(* CODESYS project FirstSteps.project

Project tree, tasks and I/O mapping:
  Device : CODESYS Control for Raspberry Pi SL, 3S - Smart Software Solutions GmbH, version 3.5.12.30
    application Application
      libraries: AC_ModuleBase, 3.5.0.0 (3S - Smart Software Solutions GmbH); Standard, 3.5.12.0 (System)
      task AC_RMP_Task (cyclic, interval t#20ms, priority 30) calls AC_PRG_RMP
      task STANDARD (cyclic, interval t#10ms, priority 5) calls AC_CALL_STANDARD_START, AC_CALL_STANDARD_END
      global variables GVL_Simulation_I_O
      AC_Std/
        global variables GVL_Room
        global variables MODULE_INFOS
        global variables GVL_MODULE_TREE
        function AC_InitInternal [ST]
        function AC_Init [ST]
        function AC_OnlineChange [ST]
        function AC_Io_ChannelRefCode_STANDARD [ST]
        program AC_CALL_STANDARD_START [ST]
        program AC_CALL_STANDARD_END [ST]
      AC_FBs/
        function block AC_Room_Light1 [ST]
        function block AC_Room_LightSimple1 [ST]
        function block AC_Room_Light2 [ST]
        function block AC_Room [ST]
      AC_RMP/
        global variables AC_RMP
        program AC_PRG_RMP [ST]
    SoftMotion General Axis Pool
    I²C
    SPI
      SPI_master : SPI master, 3S - Smart Software Solutions GmbH, version 1.0.0.0
          settings: _diBitsPerWord = 8; _diMaxSpeed = 1000000
        Monarco_HAT : Monarco HAT, Monarco.io, version 2.0.0.0
            input  Application.GVL_Room.Room.INST_Light1.INST_Switch.xIn : BOOL  // DigIn.Bit0
            input  Application.GVL_Room.Room.INST_LightSimple1.INST_SwitchSimple.xIn : BOOL  // DigIn.Bit1
            input  Application.GVL_Room.Room.INST_Light2.INST_Switch.xIn : BOOL  // DigIn.Bit2
            output Application.GVL_Room.Room.INST_LightSimple1.xSwitchedOn : BOOL  // DigOut.Bit0
            output Application.GVL_Room.Room.INST_Light1.uiBrightness : WORD  // AO0
            output Application.GVL_Room.Room.INST_Light2.uiBrightness : WORD  // AO1
            unmapped channels: DigIn, AI0, AI1, DigOut
    GPIOs_A_B : GPIOs A/B, 3S - Smart Software Solutions GmbH, version 3.5.11.0
        unmapped channels: digital inputs (GPIO0..GPIO31), digital outputs (GPIO0..GPIO31)
    Onewire
    Camera device
      <Empty>
  libraries: AC_ModuleBase, 3.5.0.0 (3S - Smart Software Solutions GmbH)
  5ce3da45-db07-42e7-a21c-a00fff4ed8f6|D:\Libraries\trunk\Application\ApplicationComposer\AC_Building\0.34.3.5 draft\floor32.bmp
  5ce3da45-db07-42e7-a21c-a00fff4ed8f6|C:\Users\Public\Pictures\Sample Pictures\Chrysanthemum.jpg
  5ce3da45-db07-42e7-a21c-a00fff4ed8f6|C:\Users\Public\Pictures\Sample Pictures\Desert.jpg
  Room
    Lights (Lights)
      Light2
        Switch (Switch)
        Switch
      LightSimple1
        SwitchSimple
        Switch (SwitchSimple)
      Light1
        Switch (Switch)
        Switch
  AC_GENERATOR_DATA
  5ce3da45-db07-42e7-a21c-a00fff4ed8f6|C:\Users\b.joedicke\Pictures\light_16.png
  5ce3da45-db07-42e7-a21c-a00fff4ed8f6|C:\Users\b.joedicke\Pictures\light_32.png
  5ce3da45-db07-42e7-a21c-a00fff4ed8f6|C:\Users\b.joedicke\Pictures\room16.bmp
  5ce3da45-db07-42e7-a21c-a00fff4ed8f6|C:\Users\b.joedicke\Pictures\room32.bmp
  5ce3da45-db07-42e7-a21c-a00fff4ed8f6|C:\Users\b.joedicke\Pictures\switch_16.png
  5ce3da45-db07-42e7-a21c-a00fff4ed8f6|C:\Users\b.joedicke\Pictures\switch_32.png
  5ce3da45-db07-42e7-a21c-a00fff4ed8f6|C:\Users\b.joedicke\Pictures\switchsimple_32.png
  5ce3da45-db07-42e7-a21c-a00fff4ed8f6|C:\room16.bmp
  5ce3da45-db07-42e7-a21c-a00fff4ed8f6|C:\Users\b.joedicke\Pictures\lightsimple_16.png
  5ce3da45-db07-42e7-a21c-a00fff4ed8f6|C:\switchsimple_16.png
  5ce3da45-db07-42e7-a21c-a00fff4ed8f6|C:\Users\b.joedicke\Pictures\switchsimple_16.png
  5ce3da45-db07-42e7-a21c-a00fff4ed8f6|C:\Users\b.joedicke\Pictures\lightsimple_32.png
  5ce3da45-db07-42e7-a21c-a00fff4ed8f6|D:\Libraries\trunk\Application\ApplicationComposer\AC_Building\0.34.3.5 draft\SwitchOnOff32.ico
  5ce3da45-db07-42e7-a21c-a00fff4ed8f6|C:\light_16.png
  5ce3da45-db07-42e7-a21c-a00fff4ed8f6|C:\light_32.png
  5ce3da45-db07-42e7-a21c-a00fff4ed8f6|D:\Libraries\trunk\Application\ApplicationComposer\AC_Building\0.34.3.5 draft\LightStandard16.ico
  5ce3da45-db07-42e7-a21c-a00fff4ed8f6|D:\Libraries\trunk\Application\ApplicationComposer\AC_Building\0.34.3.5 draft\LightStandard32.bmp
  5ce3da45-db07-42e7-a21c-a00fff4ed8f6|D:\Libraries\trunk\Application\ApplicationComposer\AC_Building\0.34.3.5 draft\LightStandard32.ico
  5ce3da45-db07-42e7-a21c-a00fff4ed8f6|D:\Libraries\trunk\Application\ApplicationComposer\AC_Building\0.34.3.5 draft\LightDimmed16.ico
  5ce3da45-db07-42e7-a21c-a00fff4ed8f6|D:\Libraries\trunk\Application\ApplicationComposer\AC_Building\0.34.3.5 draft\LightDimmed32.ico
  5ce3da45-db07-42e7-a21c-a00fff4ed8f6|D:\Libraries\trunk\Application\ApplicationComposer\AC_Building\0.34.3.5 draft\room16.bmp
  5ce3da45-db07-42e7-a21c-a00fff4ed8f6|D:\Libraries\trunk\Application\ApplicationComposer\AC_Building\0.34.3.5 draft\room32.bmp
  5ce3da45-db07-42e7-a21c-a00fff4ed8f6|D:\Libraries\trunk\Application\ApplicationComposer\AC_Building\0.34.3.5 draft\SwitchPush16.ico
  5ce3da45-db07-42e7-a21c-a00fff4ed8f6|D:\Libraries\trunk\Application\ApplicationComposer\AC_Building\0.34.3.5 draft\SwitchPush32.ico
  5ce3da45-db07-42e7-a21c-a00fff4ed8f6|D:\Libraries\trunk\Application\ApplicationComposer\AC_Building\0.34.3.5 draft\SwitchOnOff16.ico
  Room/
    text Room
    function block Room [ST]
    text list TL
    Light/
      interface ILight
      text Light
      function block Light [ST]: CallPrioMediumStart
      text LightSimple
      function block LightSimple [ST]: CallPrioMediumStart
    Switch/
      text Switch
      interface ISwitch: Push, PushLong
      function block Switch [ST]: Push, PushLong, CallPrioMediumStart
      interface ISwitchSimple: On
      text SwitchSimple
      function block SwitchSimple [ST]: On
    image pool IP
  5ce3da45-db07-42e7-a21c-a00fff4ed8f6|D:\Libraries\trunk\Application\ApplicationComposer\AC_Building\0.34.3.5 draft\room16.bmp
  5ce3da45-db07-42e7-a21c-a00fff4ed8f6|D:\Libraries\trunk\Application\ApplicationComposer\AC_Building\0.34.3.5 draft\room32.bmp
  5ce3da45-db07-42e7-a21c-a00fff4ed8f6|D:\Libraries\trunk\Application\ApplicationComposer\AC_Building\0.34.3.5 draft\SwitchPush16.ico
  5ce3da45-db07-42e7-a21c-a00fff4ed8f6|D:\Libraries\trunk\Application\ApplicationComposer\AC_Building\0.34.3.5 draft\SwitchPush32.ico
  5ce3da45-db07-42e7-a21c-a00fff4ed8f6|D:\Libraries\trunk\Application\ApplicationComposer\AC_Building\0.34.3.5 draft\LightDimmed16.ico
  5ce3da45-db07-42e7-a21c-a00fff4ed8f6|D:\Libraries\trunk\Application\ApplicationComposer\AC_Building\0.34.3.5 draft\LightDimmed32.ico
  5ce3da45-db07-42e7-a21c-a00fff4ed8f6|D:\Libraries\trunk\Application\ApplicationComposer\AC_Building\0.34.3.5 draft\LightStandard16.ico
  5ce3da45-db07-42e7-a21c-a00fff4ed8f6|D:\Libraries\trunk\Application\ApplicationComposer\AC_Building\0.34.3.5 draft\LightStandard32.ico
  5ce3da45-db07-42e7-a21c-a00fff4ed8f6|D:\Libraries\trunk\Application\ApplicationComposer\AC_Building\0.34.3.5 draft\SwitchOnOff16.ico
  5ce3da45-db07-42e7-a21c-a00fff4ed8f6|D:\Libraries\trunk\Application\ApplicationComposer\AC_Building\0.34.3.5 draft\SwitchOnOff32.ico
*)

// Device/Application/GVL_Simulation_I_O
VAR_GLOBAL

//these variables are normally real inputs and outputs. 
///For simulation reason, they are declared here and can be used to test the app.	

	xPushSwitch			: BOOL;
	xPushSimpleSwitch	: BOOL;

	uiBrightness		: UINT;
	xSimpleOn			: BOOL;
END_VAR

// Device/Application/AC_Std/GVL_Room
//Code generated by Application Composer.
//Modifying generated code is not recommended!

VAR_GLOBAL
	Room: AC_Room;
END_VAR

// Device/Application/AC_Std/MODULE_INFOS
//Code generated by Application Composer.
//Modifying generated code is not recommended!
{attribute 'global_init_slot' := '40000'}
{attribute 'init_on_onlchange'}

VAR_GLOBAL
	{attribute 'init_on_onlchange'}
	Room_INFO: AC.ModuleInfo := (pbyModuleType := ADR('Room'));
	{attribute 'init_on_onlchange'}
	Light_INFO: AC.ModuleInfo := (pbyModuleType := ADR('Light'));
	{attribute 'init_on_onlchange'}
	LightSimple_INFO: AC.ModuleInfo := (pbyModuleType := ADR('LightSimple'));
	{attribute 'init_on_onlchange'}
	Switch_INFO: AC.ModuleInfo := (pbyModuleType := ADR('Switch'));
	{attribute 'init_on_onlchange'}
	SwitchSimple_INFO: AC.ModuleInfo := (pbyModuleType := ADR('SwitchSimple'));
END_VAR

// Device/Application/AC_Std/GVL_MODULE_TREE
//Code generated by Application Composer.
//Modifying generated code is not recommended!

VAR_GLOBAL
	Module_Tree: AC.ModuleTree;
	aNodes: ARRAY[0..7] OF AC.MNode;
	AC_Environment: AC.MEnv;
END_VAR

// Device/Application/AC_RMP/AC_RMP
//Code generated by Application Composer.
//Modifying generated code is not recommended!
{attribute 'global_init_slot' := '60000'}
{attribute 'init_on_onlchange'}

VAR_GLOBAL
	{attribute 'init_on_onlchange'}
	AC_RMP_Service: AC.RMPService := (uiLocalAppID:=9744, uiNumberOfConnections:=0, pSendConnection:=0, pReceiveConnection:=0);
END_VAR

// Device/Application/AC_RMP/AC_PRG_RMP
//Code generated by Application Composer.
//Modifying generated code is not recommended!
PROGRAM AC_PRG_RMP
VAR
    itfRmpService2 : AC.IRmpService2 := 0;
    xStartCyclicAction : BOOL;
    xIsActionOngoing : BOOL;
    xValid : BOOL;
    xValidEnd : BOOL := TRUE;
END_VAR

//Code generated by Application Composer.
//Modifying generated code is not recommended!
__QUERYINTERFACE(AC_RMP_Service, itfRmpService2);
IF itfRmpService2 <> 0 AND xValidEnd THEN
    xValid := itfRmpService2.GetIsActionOngoing(xIsActionOngoing=>xIsActionOngoing);
    IF NOT xValid OR (xValid AND xIsActionOngoing) THEN
        xStartCyclicAction := FALSE;
    ELSE
        xStartCyclicAction := itfRmpService2.SetIsActionOngoing(TRUE);
    END_IF
ELSE
    xStartCyclicAction := TRUE;
END_IF
IF xStartCyclicAction THEN
    AC_RMP_Service.CyclicCall() ;
END_IF
IF itfRmpService2 <> 0 AND (xStartCyclicAction OR NOT xValidEnd) THEN
    xValidEnd := itfRmpService2.SetIsActionOngoing(FALSE);
END_IF

END_PROGRAM

// Device/Application/AC_Std/AC_CALL_STANDARD_START
//Code generated by Application Composer.
//Modifying generated code is not recommended!
PROGRAM AC_CALL_STANDARD_START

//Code generated by Application Composer.
//Modifying generated code is not recommended!
AC_Io_ChannelRefCode_STANDARD() ;
Room.CallPrioMEDIUMStart() ;

END_PROGRAM

// Device/Application/AC_Std/AC_Io_ChannelRefCode_STANDARD
//Code generated by Application Composer.
//Modifying generated code is not recommended!
FUNCTION AC_Io_ChannelRefCode_STANDARD

//Code generated by Application Composer.
//Modifying generated code is not recommended!

//Special code to make sure mapped I/O variables are updated in the correct task

{IF defined(variable:Application.GVL_Room.Room.INST_Light1.uiBrightness) AND defined(variable:Application.GVL_Room.Room.INST_LightSimple1.xSwitchedOn) AND defined(variable:Application.GVL_Room.Room.INST_Light2.uiBrightness) AND defined(variable:Application.GVL_Room.Room.INST_Light1.INST_Switch.xIn) AND defined(variable:Application.GVL_Room.Room.INST_LightSimple1.INST_SwitchSimple.xIn) AND defined(variable:Application.GVL_Room.Room.INST_Light2.INST_Switch.xIn)}
 ;
{END_IF}

END_FUNCTION

// Room/Room
FUNCTION_BLOCK Room EXTENDS AC.Module
VAR_INPUT
	//Submodule Lights
	pLights				: POINTER TO ILight;
	uiNumberOfLights	: UINT;
END_VAR
VAR_OUTPUT
END_VAR
VAR
END_VAR

END_FUNCTION_BLOCK

// Room/Light/ILight
INTERFACE ILight EXTENDS AC.IModule

END_INTERFACE

// Device/Application/AC_Std/AC_CALL_STANDARD_END
//Code generated by Application Composer.
//Modifying generated code is not recommended!
PROGRAM AC_CALL_STANDARD_END

//Code generated by Application Composer.
//Modifying generated code is not recommended!
Room.CallPrioMEDIUMEnd() ;

END_PROGRAM

// Room/Light/Light
FUNCTION_BLOCK Light EXTENDS AC.Module IMPLEMENTS ILight
VAR_INPUT
	//Submodule Switch
	Switch		: ISwitch;
	
	//parameter
	uiMaxValue	: UINT := 5000 ;
	rSpeed	: REAL := 25; //percentage per second
END_VAR
VAR_OUTPUT
	uiBrightness	: UINT;
END_VAR
VAR
	rPercentageOn	: REAL; (* percentage from 0 to 1 *)
	tTaskCycle		: TIME := T#10MS;
	rDirection		: REAL := 1; (* 1 --> switch the light on --> switch it off *)
	
	xChangeDirection: BOOL; (* helper variable *)
	xChangeDirectionPush: BOOL; (* helper variable *)
	
	iState			: INT;
END_VAR

(* Called at the start of the medium priority task if one is defined.
 Note: the return value is not used.*)
METHOD CallPrioMediumStart : BOOL
VAR
	pModule: POINTER TO AC.Module;
END_VAR
SUPER^.CallPrioMediumStart();

CASE iState OF
	
	0: (* check the state of the switch *)
		IF Switch.PushLong THEN
			xChangeDirection := TRUE;
			iState := 10;
		ELSIF NOT Switch.PushLong AND xChangeDirection THEN
			xChangeDirection := FALSE;
			iState := 20;
			
		ELSIF Switch.Push THEN
			iState := 30;
			xChangeDirectionPush := TRUE;
			
		ELSIF NOT Switch.Push AND xChangeDirectionPush THEN
			xChangeDirectionPush := FALSE;
			iState := 20;
		END_IF
	
	10: (* dim function *)
		rPercentageOn := rPercentageOn + rDirection * rSpeed * TIME_TO_REAL(tTaskCycle)/100000;
		IF rPercentageOn > 1 THEN
			rPercentageOn := 1;
			
		ELSIF rPercentageOn < 0 THEN
			rPercentageOn := 0;
		END_IF
		iState := 0;
	
	20: (* check if the direction must be changed *)
		IF rDirection = 1 AND rPercentageOn = 1 THEN
			rDirection := -1;
		ELSIF
			rDirection = -1 AND rPercentageOn = 0 THEN
			rDirection := 1;
		END_IF
		iState := 0;
	
	30:(* invert light *)
		IF rPercentageOn = 1 THEN
			rPercentageOn :=0;
		ELSE
			rPercentageOn := 1;
		END_IF
		iState := 0;

END_CASE

uiBrightness := REAL_TO_UINT(rPercentageOn*uiMaxValue);
END_METHOD

END_FUNCTION_BLOCK

// Room/Switch/Switch
FUNCTION_BLOCK Switch EXTENDS AC.Module IMPLEMENTS ISwitch
VAR_INPUT
	// Input
	xIn		: BOOL;
	//parameter
	tTimer	: TIME := T#500MS;
END_VAR

VAR
	timerLong	: TON; (* timer to know how long the switch is tapped *)
	
	xPush	: BOOL; (* signal to toggle the light *)
	xPushLong : BOOL; (* signal to dim the light *)
	
	iState	: INT;
END_VAR

PROPERTY PUBLIC Push : BOOL
GET
Push := xPush;
END_GET
END_PROPERTY

PROPERTY PUBLIC PushLong : BOOL
GET
PushLong := xPushLong;
END_GET
END_PROPERTY

(* Called at the start of the medium priority task if one is defined.
 Note: the return value is not used.*)
METHOD CallPrioMediumStart : BOOL
SUPER^.CallPrioMediumStart();

xPush := FALSE;

CASE iState OF
	0: (* initialization *)
		xPush := xPushLong := FALSE;
		IF NOT xIn THEN
			iState := 10;
		END_IF
		
	10: (* switch is pushed *)
		IF xIn THEN
			iState := 20;
			timerLong(IN := FALSE, PT := tTimer);
		END_IF

	20: (* timer is started, to check if the toggle or dim function should be used *)
		timerLong(IN := TRUE);
		IF NOT xIn THEN
			xPush := TRUE;
			iState := 0;
		ELSIF timerLong.Q THEN
			iState := 30;
		END_IF
		
	30: (* the dim function is used *)
		xPushLong := TRUE;
		IF NOT xIn THEN
			iState := 0;
		END_IF
		

END_CASE
END_METHOD

END_FUNCTION_BLOCK

// Room/Switch/ISwitch
INTERFACE ISwitch IMPLEMENTS AC.IModule

PROPERTY Push : BOOL
GET
END_GET
END_PROPERTY

PROPERTY PushLong : BOOL
GET
END_GET
END_PROPERTY

END_INTERFACE

// Room/Light/LightSimple
FUNCTION_BLOCK LightSimple EXTENDS AC.Module IMPLEMENTS ILight
VAR_INPUT
	// Submodule Switch
	SwitchSimple	: ISwitchSimple;
END_VAR
VAR_OUTPUT
	xSwitchedOn		: BOOL;
END_VAR
VAR
END_VAR

(* Called at the start of the medium priority task if one is defined.
 Note: the return value is not used.*)
METHOD CallPrioMediumStart : BOOL
SUPER^.CallPrioMediumStart();

xSwitchedOn := SwitchSimple.On;
END_METHOD

END_FUNCTION_BLOCK

// Room/Switch/SwitchSimple
FUNCTION_BLOCK SwitchSimple EXTENDS AC.Module IMPLEMENTS ISwitchSimple
VAR_INPUT
	// Input
	xIn		: BOOL;
END_VAR
VAR_OUTPUT
END_VAR
VAR
	xOn	: BOOL;
END_VAR

PROPERTY PUBLIC On : BOOL
GET
On := xIn;
END_GET
END_PROPERTY

END_FUNCTION_BLOCK

// Room/Switch/ISwitchSimple
INTERFACE ISwitchSimple IMPLEMENTS AC.IModule

PROPERTY On : BOOL
GET
END_GET
END_PROPERTY

END_INTERFACE

// Device/Application/AC_FBs/AC_Room_Light1
//Code generated by Application Composer.
//Modifying generated code is not recommended!
FUNCTION_BLOCK AC_Room_Light1 EXTENDS Light
VAR_INPUT 
    INST_Switch : Switch;
END_VAR

//Code generated by Application Composer.
//Modifying generated code is not recommended!
SUPER^();

END_FUNCTION_BLOCK

// Device/Application/AC_FBs/AC_Room_LightSimple1
//Code generated by Application Composer.
//Modifying generated code is not recommended!
FUNCTION_BLOCK AC_Room_LightSimple1 EXTENDS LightSimple
VAR_INPUT 
    INST_SwitchSimple : SwitchSimple;
END_VAR

//Code generated by Application Composer.
//Modifying generated code is not recommended!
SUPER^();

END_FUNCTION_BLOCK

// Device/Application/AC_FBs/AC_Room_Light2
//Code generated by Application Composer.
//Modifying generated code is not recommended!
FUNCTION_BLOCK AC_Room_Light2 EXTENDS Light
VAR_INPUT 
    INST_Switch : Switch;
END_VAR

//Code generated by Application Composer.
//Modifying generated code is not recommended!
SUPER^();

END_FUNCTION_BLOCK

// Device/Application/AC_FBs/AC_Room
//Code generated by Application Composer.
//Modifying generated code is not recommended!
FUNCTION_BLOCK AC_Room EXTENDS Room
VAR_INPUT 
    INST_Light1 : AC_Room_Light1;
    INST_LightSimple1 : AC_Room_LightSimple1;
    INST_Light2 : AC_Room_Light2;
    AC_ARRAY_pLights : ARRAY[0..2] OF ILight;
END_VAR

//Code generated by Application Composer.
//Modifying generated code is not recommended!
SUPER^();

END_FUNCTION_BLOCK

// Device/Application/AC_Std/AC_InitInternal
//Code generated by Application Composer.
//Modifying generated code is not recommended!
FUNCTION AC_InitInternal
VAR_INPUT
  bOnlineChange : BOOL ;
END_VAR
VAR
  hnd : AC.ModuleHandle ;
END_VAR

//Code generated by Application Composer.
//Modifying generated code is not recommended!
AC_Environment.mtree := Module_Tree ;
AC_Environment.rmps := AC_RMP_Service ;
{IF defined(variable:AC_Environment.exts)}
	AC_Environment.exts := 0 ;
	AC_Environment.uiexts := 0 ;
{END_IF}
Module_Tree.Init(ADR(aNodes), 8);
hnd := Module_Tree.AddChild(0, Room);
Room.SetIdentification(ADR('Room'), ADR(Room_INFO), 16#2610A9CF, hnd, ADR(AC_Environment)) ;
hnd := Module_Tree.AddChild(Room, Room.INST_Light2);
Room.INST_Light2.SetIdentification(ADR('Light2'), ADR(Light_INFO), 16#26100F2D, hnd, ADR(AC_Environment)) ;
hnd := Module_Tree.AddChild(Room, Room.INST_LightSimple1);
Room.INST_LightSimple1.SetIdentification(ADR('LightSimple1'), ADR(LightSimple_INFO), 16#2610E8D4, hnd, ADR(AC_Environment)) ;
hnd := Module_Tree.AddChild(Room, Room.INST_Light1);
Room.INST_Light1.SetIdentification(ADR('Light1'), ADR(Light_INFO), 16#2610C045, hnd, ADR(AC_Environment)) ;
hnd := Module_Tree.AddChild(Room.INST_Light2, Room.INST_Light2.INST_Switch);
Room.INST_Light2.INST_Switch.SetIdentification(ADR('Switch'), ADR(Switch_INFO), 16#261067C5, hnd, ADR(AC_Environment)) ;
hnd := Module_Tree.AddChild(Room.INST_LightSimple1, Room.INST_LightSimple1.INST_SwitchSimple);
Room.INST_LightSimple1.INST_SwitchSimple.SetIdentification(ADR('SwitchSimple'), ADR(SwitchSimple_INFO), 16#26107A30, hnd, ADR(AC_Environment)) ;
hnd := Module_Tree.AddChild(Room.INST_Light1, Room.INST_Light1.INST_Switch);
Room.INST_Light1.INST_Switch.SetIdentification(ADR('Switch'), ADR(Switch_INFO), 16#2610E8FB, hnd, ADR(AC_Environment)) ;
Room.uiNumberOfLights := 3;
Room.AC_ARRAY_pLights[0] := Room.INST_Light1;
Room.AC_ARRAY_pLights[1] := Room.INST_LightSimple1;
Room.AC_ARRAY_pLights[2] := Room.INST_Light2;
Room.pLights := ADR(Room.AC_ARRAY_pLights);
Room.INST_Light1.Switch := Room.INST_Light1.INST_Switch;
Room.INST_LightSimple1.SwitchSimple := Room.INST_LightSimple1.INST_SwitchSimple;
Room.INST_Light2.Switch := Room.INST_Light2.INST_Switch;
IF bOnlineChange THEN
    Room.INST_Light1.uiMaxValue := 5000;
    Room.INST_Light1.rSpeed := 25;
    Room.INST_Light2.uiMaxValue := 5000;
    Room.INST_Light2.rSpeed := 25;
    Room.INST_Light1.INST_Switch.tTimer := TIME#500ms;
    Room.INST_Light2.INST_Switch.tTimer := TIME#500ms;
END_IF
Room.Init(bOnlineChange);

END_FUNCTION

// Device/Application/AC_Std/AC_Init
//Code generated by Application Composer.
//Modifying generated code is not recommended!
{attribute 'linkalways'}
{attribute 'call_after_global_init_slot' := '1234'}
FUNCTION AC_Init

//Code generated by Application Composer.
//Modifying generated code is not recommended!
AC_InitInternal(FALSE);

END_FUNCTION

// Device/Application/AC_Std/AC_OnlineChange
//Code generated by Application Composer.
//Modifying generated code is not recommended!
{attribute 'linkalways'}
{attribute 'call_after_online_change_slot' := '1234'}
FUNCTION AC_OnlineChange

//Code generated by Application Composer.
//Modifying generated code is not recommended!
Room.OnBeforeOnlineChange();
AC_InitInternal(TRUE);
Room.OnAfterOnlineChange();

END_FUNCTION

(* text list TL (id | default)
  Room_Desc | This is a room.
  UnitStandard_Task | This is a standard task.
  Role_Lights | Lights
  Light_Desc | This is a light, which can be dimmed and switched on and off.
  Switch_Desc | This is a switch, which has a tap and dim function.
  Light_Name_xOn | xOn
  Light_Desc_xOn | Licht eingeschalten (True) / ausgeschalten (False)
  Role_Switch | Switch
  Name_uiBrightness | Brightness
  Desc_uiBrightness | The brightness of the light.
  Name_uiMaxValue | maxLightValue
  Desc_uiMaxValue | The maximum value of the light.
  NAME_rSpeed | Speed
  DESC_rSpeed | The speed of the dimmer.
  NAME_tTimer | Timer
  DESC_tTimer | The time the switch has to wait before switching to the dim modus.
  Switch_Name_xIn | xIn
  Switch_Desc_xIn | Input of the Switch.
  SwitchSimple_Name_xIn | xIn (Simple)
  SwitchSimple_Desc_xIn | State of the switch (on / off)
  LightSimple_Desc | The simple light can be switched on and off.
  Name_switchedOn | SwitchedOn
  Desc_switchedOn | True, when the light is switched on and false when it is off.
  SwitchSimple_Desc | The simple switch has an on and off position.
   |  *)

(* text Room
MODULE Room IMPLEMENTED_BY Room
SEC MetaData
	Desc       := TL.Room_Desc ;
	Category   := 'FirstSteps' ;
	Icon_16    := IP.Room_Icon_16 ;
	Icon_32    := IP.Room_Icon_32 ;
END_SEC
SEC Toplevel
	GVL_name := 'GVL_%InstanceName%' ;
    SEC Standard_Task : MEDIUM
		Name  := STANDARD ;
		Desc  := TL.UnitStandard_Task ;
		Flags := CREATE_IF_MISSING | UPDATE_IOS ; ( * at least one task must use the "UPDATE_IOS" flag. * )
	END_SEC
END_SEC

SEC Slots
	SEC Slot_Multi	: Lights
		Variable	:= pLights;
		Var_Count	:= uiNumberOfLights;
		Role		:= TL.Role_Lights;
		Cardinality := [1..3];
		Type		:= SUBMODULE;
	END_SEC	
END_SEC
*)

(* text Light
MODULE Light IMPLEMENTED_BY Light
SEC MetaData
	Desc := TL.Light_Desc ;
	Category := 'FirstSteps' ;
	Icon_16 := IP.Light_Icon_16 ;
	Icon_32 := IP.Light_Icon_32 ;
END_SEC

SEC Slots
	SEC Slot : Switch
		Variable := Switch;
		Role := TL.Role_Switch;
		Type := SUBMODULE;
	END_SEC
END_SEC

SEC IO
	SEC Output : uiBrightness
		Variable := uiBrightness;
		Name := TL.Name_uiBrightness;
		Desc := TL.Desc_uiBrightness;
	END_SEC
END_SEC

SEC Parameters
	SEC Param : uiMaxValue
		Variable := uiMaxValue;
		Name := TL.Name_uiMaxValue;
		Desc := TL.Desc_uiMaxValue;
	END_SEC

	SEC Param : rSpeed
		Variable := rSpeed ;
		Name := TL.NAME_rSpeed ;
		Desc := TL.DESC_rSpeed ;
	END_SEC
END_SEC
*)

(* text LightSimple
MODULE LightSimple IMPLEMENTED_BY LightSimple
SEC MetaData
	Desc       := TL.LightSimple_Desc ;
	Category   := 'FirstSteps' ;
	Icon_16    := IP.LightSimple_Icon_16 ;
	Icon_32    := IP.LightSimple_Icon_32 ;
END_SEC

SEC Slots
	SEC Slot : SwitchSimple
		Variable := SwitchSimple;
		Role := TL.Role_Switch;
		Type := SUBMODULE;
	END_SEC
END_SEC

SEC IO
	SEC Output : SwitchedOn
		Variable := xSwitchedOn;
		Name := TL.Name_switchedOn;
		Desc := TL.Desc_switchedOn;
	END_SEC
END_SEC
*)

(* text Switch
MODULE Switch IMPLEMENTED_BY Switch
SEC MetaData
	Desc       := TL.Switch_Desc;
	Category   := 'FirstSteps';
	Icon_16    := IP.Switch_Icon_16;
	Icon_32    := IP.Switch_Icon_32;
END_SEC

SEC Parameters
	SEC Param : tTimer
		Variable := tTimer;
		Name := TL.NAME_tTimer;
		Desc := TL.DESC_tTimer;
	END_SEC
END_SEC

SEC IO
	SEC Input : xIn
		Variable := xIn;
		Name := TL.Switch_Name_xIn;
		Desc := TL.Switch_Desc_xIn;
	END_SEC

END_SEC
*)

(* text SwitchSimple
MODULE SwitchSimple IMPLEMENTED_BY SwitchSimple
    SEC MetaData
        Desc := TL.SwitchSimple_Desc ;
        Category := 'FirstSteps' ;
        Icon_16 := IP.SwitchSimple_Icon_16 ;
        Icon_32 := IP.SwitchSimple_Icon_32 ;
    END_SEC
    
SEC IO
	SEC Input : xIn
		Variable := xIn;
		Name := TL.SwitchSimple_Name_xIn;
		Desc := TL.SwitchSimple_Desc_xIn;
	END_SEC
END_SEC
*)
